// TIA Portal project "Practica_7_p3" (V14)

(* hardware
DEVICE "S7-1200 station_1"  S7-1200 Station
   slot 0: "Rack_0"  S7-1200 Rack  Rack  V1.0
   slot 1: "PLC_1"  CPU 1214C DC/DC/DC  6ES7 214-1AG40-0XB0  V4.2
*)

// ===== PLC "PLC_1"  CPU 1214C DC/DC/DC =====

VAR_GLOBAL   // PLC tag table "Default tag table"
   "APAGADO" AT %M0.0 : Bool;
   "Y" AT %M0.1 : Bool;
   "R" AT %M0.2 : Bool;
   "G" AT %M0.3 : Bool;
   "S" AT %M0.4 : Bool;
   "LUZ_AMARILLA" AT %Q0.0 : Bool;
   "LUZ_ROJA" AT %Q0.1 : Bool;
   "LUZ_VERDE" AT %Q0.2 : Bool;
   "PM" AT %I0.0 : Bool;
   "PP" AT %I0.1 : Bool;
   "ENABLE" AT %M0.5 : Bool;
END_VAR

DATA_BLOCK "DB_TIMERS_CONFIG"   // DB4
{ S7_Optimized_Access := 'TRUE' }
VERSION : 0.1
   VAR
      TA : Time := T#6s;
      TV : Time := T#5s;
      TR : Time := T#5s;
   END_VAR
BEGIN
END_DATA_BLOCK

// folder: System blocks/Program resources

DATA_BLOCK "t_a"   // DB1
{ S7_Optimized_Access := 'TRUE' }
AUTHOR : Simatic
FAMILY : IEC
NAME : IEC_TMR
VERSION : 1.0
// stored: InstanceOfName IEC_TIMER
"IEC_TIMER"
BEGIN
END_DATA_BLOCK

DATA_BLOCK "t_r"   // DB2
{ S7_Optimized_Access := 'TRUE' }
AUTHOR : Simatic
FAMILY : IEC
NAME : IEC_TMR
VERSION : 1.0
// stored: InstanceOfName IEC_TIMER
"IEC_TIMER"
BEGIN
END_DATA_BLOCK

DATA_BLOCK "t_v"   // DB3
{ S7_Optimized_Access := 'TRUE' }
AUTHOR : Simatic
FAMILY : IEC
NAME : IEC_TMR
VERSION : 1.0
// stored: InstanceOfName IEC_TIMER
"IEC_TIMER"
BEGIN
END_DATA_BLOCK

// folder: (top level)

FUNCTION "SEMAFORO_V2" : Void   // FC1, LAD
{ S7_Optimized_Access := 'TRUE' }
VERSION : 0.1
   VAR_INPUT
      ENABLE : Bool;
      TA : Time;
      TV : Time;
      TR : Time;
   END_VAR
   VAR_OUTPUT
      LA : Bool;
      LR : Bool;
      LV : Bool;
   END_VAR
   VAR_TEMP   // added for the SCL form of the ladder/FBD networks
      _w1 : Bool;
      _w2 : Bool;
      _w3 : Bool;
      _w4 : Bool;
   END_VAR
BEGIN

REGION Network 1
   // INICIALIZACIÓN
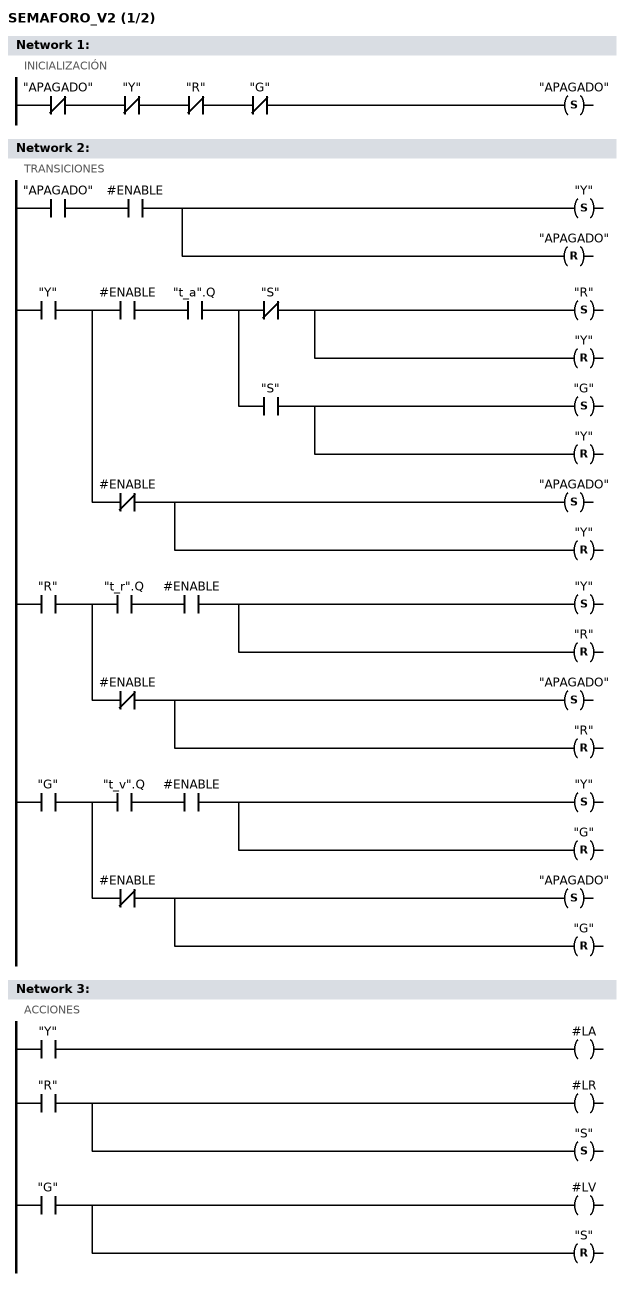
   RUNG wire#powerrail
      I_Contact( "APAGADO" )
      I_Contact( "Y" )
      I_Contact( "R" )
      I_Contact( "G" )
      S_Coil( "APAGADO" )
   END_RUNG
   // the same network as SCL:
   IF NOT "APAGADO" AND NOT "Y" AND NOT "R" AND NOT "G" THEN "APAGADO" := TRUE; END_IF;
END_REGION

REGION Network 2
   // TRANSICIONES
   RUNG wire#powerrail
      Contact( "APAGADO" )
      Contact( #ENABLE )
      wire#w1
      S_Coil( "Y" )
   END_RUNG
   RUNG wire#w1
      R_Coil( "APAGADO" )
   END_RUNG
   RUNG wire#powerrail
      Contact( "Y" )
      wire#w2
      Contact( #ENABLE )
      Contact( "t_a".Q )
      wire#w3
      I_Contact( "S" )
      wire#w4
      S_Coil( "R" )
   END_RUNG
   RUNG wire#w4
      R_Coil( "Y" )
   END_RUNG
   RUNG wire#w3
      Contact( "S" )
      wire#w5
      S_Coil( "G" )
   END_RUNG
   RUNG wire#w5
      R_Coil( "Y" )
   END_RUNG
   RUNG wire#w2
      I_Contact( #ENABLE )
      wire#w6
      S_Coil( "APAGADO" )
   END_RUNG
   RUNG wire#w6
      R_Coil( "Y" )
   END_RUNG
   RUNG wire#powerrail
      Contact( "R" )
      wire#w7
      Contact( "t_r".Q )
      Contact( #ENABLE )
      wire#w8
      S_Coil( "Y" )
   END_RUNG
   RUNG wire#w8
      R_Coil( "R" )
   END_RUNG
   RUNG wire#w7
      I_Contact( #ENABLE )
      wire#w9
      S_Coil( "APAGADO" )
   END_RUNG
   RUNG wire#w9
      R_Coil( "R" )
   END_RUNG
   RUNG wire#powerrail
      Contact( "G" )
      wire#w10
      Contact( "t_v".Q )
      Contact( #ENABLE )
      wire#w11
      S_Coil( "Y" )
   END_RUNG
   RUNG wire#w11
      R_Coil( "G" )
   END_RUNG
   RUNG wire#w10
      I_Contact( #ENABLE )
      wire#w12
      S_Coil( "APAGADO" )
   END_RUNG
   RUNG wire#w12
      R_Coil( "G" )
   END_RUNG
   // the same network as SCL:
   IF "APAGADO" AND #ENABLE THEN
       "Y" := TRUE;
       "APAGADO" := FALSE;
   END_IF;
   #_w1 := "Y" AND #ENABLE AND "t_a".Q;
   IF #_w1 AND NOT "S" THEN "R" := TRUE; END_IF;
   #_w2 := "Y";
   IF #_w1 AND NOT "S" THEN "Y" := FALSE; END_IF;
   IF #_w1 AND "S" THEN
       "G" := TRUE;
       "Y" := FALSE;
   END_IF;
   IF #_w2 AND NOT #ENABLE THEN
       "APAGADO" := TRUE;
       "Y" := FALSE;
   END_IF;
   IF "R" AND "t_r".Q AND #ENABLE THEN "Y" := TRUE; END_IF;
   #_w3 := "R";
   IF "R" AND "t_r".Q AND #ENABLE THEN "R" := FALSE; END_IF;
   IF #_w3 AND NOT #ENABLE THEN
       "APAGADO" := TRUE;
       "R" := FALSE;
   END_IF;
   IF "G" AND "t_v".Q AND #ENABLE THEN "Y" := TRUE; END_IF;
   #_w4 := "G";
   IF "G" AND "t_v".Q AND #ENABLE THEN "G" := FALSE; END_IF;
   IF #_w4 AND NOT #ENABLE THEN
       "APAGADO" := TRUE;
       "G" := FALSE;
   END_IF;
END_REGION

REGION Network 3
   // ACCIONES
   RUNG wire#powerrail
      Contact( "Y" )
      Coil( #LA )
   END_RUNG
   RUNG wire#powerrail
      Contact( "R" )
      wire#w1
      Coil( #LR )
   END_RUNG
   RUNG wire#w1
      S_Coil( "S" )
   END_RUNG
   RUNG wire#powerrail
      Contact( "G" )
      wire#w2
      Coil( #LV )
   END_RUNG
   RUNG wire#w2
      R_Coil( "S" )
   END_RUNG
   // the same network as SCL:
   #LA := "Y";
   #LR := "R";
   IF "R" THEN "S" := TRUE; END_IF;
   #LV := "G";
   IF "G" THEN "S" := FALSE; END_IF;
END_REGION

REGION Network 4
   // TIMERS Y CONTADORES
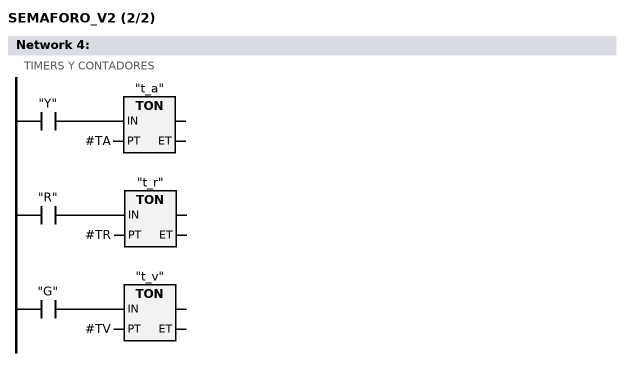
   "t_a".TON(IN := "Y", PT := #TA);
   "t_r".TON(IN := "R", PT := #TR);
   "t_v".TON(IN := "G", PT := #TV);
END_REGION
END_FUNCTION

ORGANIZATION_BLOCK "Main"   // OB1, LAD, ProgramCycle
TITLE = "Main Program Sweep (Cycle)"
{ S7_Optimized_Access := 'TRUE' }
VERSION : 0.1
   VAR_INPUT
      Initial_Call : Bool;   // Initial call of this OB
      Remanence : Bool;   // =True, if remanent data are available
   END_VAR
BEGIN

REGION Network 1
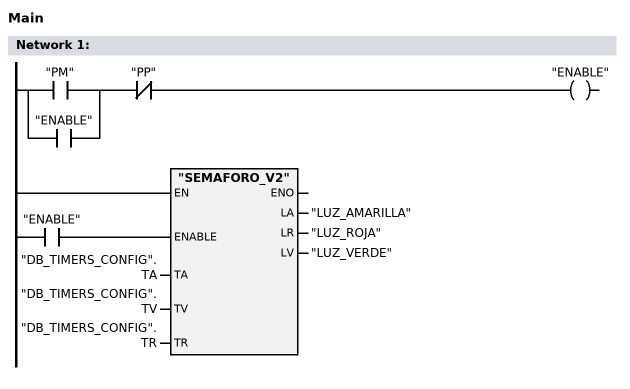
   RUNG wire#powerrail
      Contact( "PM" )
      wire#w1
      I_Contact( "PP" )
      Coil( "ENABLE" )
   END_RUNG
   RUNG wire#powerrail
      Contact( "ENABLE" )
   END_RUNG wire#w1
   RUNG wire#powerrail
      "SEMAFORO_V2"(ENABLE := wire#w2, TA := "DB_TIMERS_CONFIG".TA, TV := "DB_TIMERS_CONFIG".TV, TR := "DB_TIMERS_CONFIG".TR, LA => "LUZ_AMARILLA", LR => "LUZ_ROJA", LV => "LUZ_VERDE")
   END_RUNG
   RUNG wire#powerrail
      Contact( "ENABLE" )
   END_RUNG wire#w2
   // the same network as SCL:
   "ENABLE" := ("PM" OR "ENABLE") AND NOT "PP";
   "SEMAFORO_V2"(ENABLE := "ENABLE",
                 TA := "DB_TIMERS_CONFIG".TA,
                 TV := "DB_TIMERS_CONFIG".TV,
                 TR := "DB_TIMERS_CONFIG".TR,
                 LA => "LUZ_AMARILLA",
                 LR => "LUZ_ROJA",
                 LV => "LUZ_VERDE");
END_REGION
END_ORGANIZATION_BLOCK